(*
SPDX-FileCopyrightText: © 2026 Oleksandr Tiutyk <trofimich@gmail.com>
SPDX-License-Identifier: MIT
License: https://opensource.org/license/mit
*)

(*!
<summary>Marker interface for composite activities that coordinate one or more child activities.</summary>
*)

INTERFACE ICompositeActivity EXTENDS IActivity

END_INTERFACE

(* stored: Version 1.1.0.1
   Itf ICompositeActivity: Id {dd4eb94d-0fc9-4489-9a38-813858f781f6} *)
